{attribute 'linkalways'} 
{attribute 'no_explicit_call' := 'This FB is a CLASS and must be accessed using methods or properties'}
{attribute 'enable_dynamic_creation'}
FUNCTION_BLOCK JsonDeserializerNullObjectForwardEnumerator EXTENDS Disposable IMPLEMENTS I_DeserializerObjectForwardEnumerator, I_EventHandler
VAR
	parent : I_JsonDeserializer;
	nullNode : I_Deserializer;
	invalid : BOOL := FALSE; 
END_VAR

PROPERTY PUBLIC Current : I_Deserializer
GET
Current := nullNode;
END_GET
END_PROPERTY

METHOD FB_exit : BOOL
VAR_INPUT
	bInCopyCode : BOOL; // if TRUE, the exit method is called for exiting an instance that is copied afterwards (online change).
END_VAR
IF bInCopyCode THEN
	RETURN;
END_IF

IF parent = 0 THEN
	RETURN;
END_IF

parent.OffEvent('OnChanged',THIS^);
parent.OffEvent('OnDisposed',THIS^);
END_METHOD

METHOD FB_init : BOOL
VAR_INPUT
	bInitRetains : BOOL; // if TRUE, the retain variables are initialized (warm start / cold start)
	bInCopyCode : BOOL;  // if TRUE, the instance afterwards gets moved into the copy code (online change)
	ParentJsonDeserializer : I_JsonDeserializer;
	ParentNullDeserializer : I_Deserializer;
END_VAR
parent := ParentJsonDeserializer;
nullNode := ParentNullDeserializer;

parent.OnEvent('OnChanged',THIS^);
parent.OnEvent('OnDisposed',THIS^);
END_METHOD

METHOD PUBLIC HandleEvent
VAR_INPUT
	Event : I_Event;
END_VAR
VAR
	changedEvent : I_JsonDeserializerChangedEvent;
	disposedEvent : I_JsonDeserializerDisposedEvent;
END_VAR
IF __QUERYINTERFACE(Event, changedEvent) THEN
	invalid := TRUE;
ELSIF __QUERYINTERFACE(Event, disposedEvent) THEN
	parent := 0;
	Dispose();
END_IF
END_METHOD

PROPERTY PUBLIC IsValid : BOOL
GET // PUBLIC
IsValid := (NOT invalid AND parent <> 0);
END_GET
END_PROPERTY

PROPERTY Key : T_MAXSTRING
GET
END_GET
END_PROPERTY

METHOD PUBLIC MoveNext : BOOL
MoveNext := FALSE;
END_METHOD

END_FUNCTION_BLOCK

(* stored: Version 1.1.0.1, ProductVersion 3.1.4024.12
   POU JsonDeserializerNullObjectForwardEnumerator: Id {de607b30-c508-4750-ac61-6c34349c7101}, SpecialFunc None
   Folder Constructor: Id {19d72c4b-e6cc-4fa9-b350-d7c1c306e1f3}
   Folder Destructor: Id {ef69be40-784e-4430-a130-2c09f1a16cad}
   Property Current: Id {18634c32-8dec-403e-8daa-75ced10f09e9}
   Get Get: Id {5dddd4e5-565e-46a7-aeac-61a2406afe33}
   Method FB_exit: Id {edcd2e4c-61d9-4d2f-b512-21b5912689f6}
   Method FB_init: Id {593563c1-6ea6-4950-a46c-59ba3fc44d33}
   Method HandleEvent: Id {779a0f76-4de5-4016-82ca-9c6379b50d4e}
   Property IsValid: Id {1af8eb32-e8f7-4775-b07d-66c710eb7b12}
   Get Get: Id {197cf698-28a5-4a23-9fa5-35fcf06beb4c}
   Property Key: Id {4eabe5db-a8a4-4733-a319-f5d31154dc40}
   Get Get: Id {ba522038-81ff-4bd2-9b5a-a1f7cd4b316d}
   Method MoveNext: Id {27f0f1ae-e691-43e5-b7b7-997e6c2c8683} *)
